KUKA KRL program: chk_w5_grp3_opn.src, chk_w5_grp3_opn.dat

--- chk_w5_grp3_opn.src ---
&ACCESS RVO4
&REL 6
&COMMENT Check grp Z3 abertos AXOR
&PARAM TEMPLATE = C:\KRC\Roboter\Template\vorgabe
&PARAM EDITMASK = *
DEF chk_w5_grp3_opn( )
;FOLD ; Programa de verificacao de grampos Z3 aberto AXOR;%{PE}%R 4.1.16,%MKUKATPBASIS,%CCOMMENT,%VNORMAL,%P 2:Programa de verificacao de grampos Z3 aberto AXOR
;ENDFOLD

$TIMER[10] = 0
$TIMER_STOP[10] = FALSE

;FOLD WAIT FOR ( IN 495 'Z3.1 ABERTO' );%{PE}%R 8.2.24,%MKUKATPBASIS,%CEXT_WAIT_FOR,%VEXT_WAIT_FOR,%P 2:, 4:, 5:$IN, 6:495, 7:Z3.1 ABERTO, 9:
WAIT FOR  ( $IN[495] )
;ENDFOLD
;FOLD WAIT FOR ( IN 513 'Z3.2 ABERTO' );%{PE}%R 8.2.24,%MKUKATPBASIS,%CEXT_WAIT_FOR,%VEXT_WAIT_FOR,%P 2:, 4:, 5:$IN, 6:513, 7:Z3.2 ABERTO, 9:
WAIT FOR  ( $IN[513] )
;ENDFOLD
;FOLD WAIT FOR ( NOT IN 496 'Z3.1 FECHADO' );%{PE}%R 8.2.24,%MKUKATPBASIS,%CEXT_WAIT_FOR,%VEXT_WAIT_FOR,%P 2:, 4:NOT, 5:$IN, 6:496, 7:Z3.1 FECHADO, 9:
WAIT FOR  (  NOT $IN[496] )
;ENDFOLD
;FOLD WAIT FOR ( NOT IN 514 'Z3.2 FECHADO' );%{PE}%R 8.2.24,%MKUKATPBASIS,%CEXT_WAIT_FOR,%VEXT_WAIT_FOR,%P 2:, 4:NOT, 5:$IN, 6:514, 7:Z3.2 FECHADO, 9:
WAIT FOR  (  NOT $IN[514] )
;ENDFOLD

$TIMER_STOP[10] = TRUE
$TIMER[10] = 0

END

--- chk_w5_grp3_opn.dat ---
&ACCESS RVO4
&REL 6
&COMMENT Check grp Z3 abertos AXOR
&PARAM TEMPLATE = C:\KRC\Roboter\Template\vorgabe
&PARAM EDITMASK = *
DEFDAT chk_w5_grp3_opn
;FOLD EXTERNAL DECLARATIONS;%{PE}%V3.2.0,%MKUKATPBASIS,%CEXT,%VCOMMON,%P
;FOLD BAS EXT;%{PE}%V3.2.0,%MKUKATPBASIS,%CEXT,%VEXT,%P
EXT  BAS (BAS_COMMAND  :IN,REAL  :IN )
DECL INT SUCCESS
;ENDFOLD
;FOLD GRIPPER EXT;%{E}%V3.2.0,%MKUKATPGRIPPER,%CEXT,%VEXT,%P
EXT  H50 (INT:IN, INT:IN ,INT:IN ,GRP_TYP:IN)
;ENDFOLD
;FOLD SPOT EXT;%{E}%V3.2.0,%MKUKATPSPOT,%CEXT,%VEXT,%P
EXT  USERSPOT (S_COMMAND  :IN, SPOT_TYPE:IN)
;ENDFOLD
;FOLD USER EXT;%{E}%V3.2.0,%MKUKATPUSER,%CEXT,%VEXT,%P
;Make here your modifications
;ENDFOLD
;ENDFOLD

ENDDAT
